// TIA Portal V21 export
DATA_BLOCK "DB604"   // DB604
TITLE = DB604
AUTHOR : PRECISE
FAMILY : PRECISE
// CIP FILLING
// stored: AutoNumber false, InstanceOfName FB604, InstanceOfType FB
"FB604"
   // VAR_INPUT
   //    CipSelected : Bool;
   //    CycleEnable : Bool;
   //    CycleRunning : Bool;
   //    SecPulse : Bool;
   //    AlwaysTrue : Bool;
   //    ActualQuantity : Real;
   //    ActualConductivity : Real;
   //    DrainWeight : Real;
   //    ActualRepetition : Int;
   //    ParaIn { ExternalAccessible := 'False'; ExternalVisible := 'False'; ExternalWritable := 'False'} : "FillingInputs";
   // END_VAR
   // VAR_OUTPUT
   //    Started : Bool;
   //    SWZDV : Bool;
   //    PWZDV : Bool;
   //    WFIZDV : Bool;
   //    RinsePump : Bool;
   //    ParaOut : "FillingOutputs";
   //    FillTimeMinPV : DInt;
   //    FillTimeSecPV : DInt;
   //    PulsingTimePV : Int;
   //    RinseTimePV : Int;
   //    StepStatus : String[60];
   //    Print : "FillingPrint";
   //    Print_1 : "PulsingPrint";
   // END_VAR
   // VAR_IN_OUT
   //    Over : Bool;
   //    OverTemp : Bool;
   //    LineValvesTemp : Bool;
   //    ZDVTemp : Bool;
   //    PulsingValveTemp : Bool;
   //    ActualFillQuantity : Real;
   //    FillQuantityToleranceCalc : Real;
   //    Temp1 : Int;
   //    Temp2 : Int;
   //    SampledConductivity : Real;
   //    ConductivitySuccess : Bool;
   //    RE1 : Bool;
   //    RE2 : Bool;
   //    RE3 : Bool;
   //    LineValves : Bool;
   // END_VAR
   // VAR
   //    ValveOnDelayPV : Int;
   //    ValveOffDelayPV : Int;
   //    FillTimer { S7_SetPoint := 'True'} : "FB101";
   //    "Pulsing/Rinsing" { S7_SetPoint := 'True'} : "FB102";
   //    StepDelay { S7_SetPoint := 'True'} : "FB110";
   //    ResetPrintValues { S7_SetPoint := 'True'} : TON_TIME;
   // END_VAR
BEGIN
END_DATA_BLOCK
